# EPICS substitutions: MOXA12XX/MOXA12XX-IOC-01App/Db/moxa_e1242_misc.substitutions
file "moxa_e1242_misc.template" {

pattern {NAME, P, ASYNPORT, CHAN}
{"\$(NAME)", "\$(P)", "\$(ASYNPORT)", "0"}
{"\$(NAME)", "\$(P)", "\$(ASYNPORT)", "1"}
{"\$(NAME)", "\$(P)", "\$(ASYNPORT)", "2"}
{"\$(NAME)", "\$(P)", "\$(ASYNPORT)", "3"}
}
